TYPE ST_OutputStationHSSustainabilityData :
STRUCT
	{attribute 'OPC.UA.DA.Description' := 'Dummy (for making struct visible on OPC UA'}
	bDummy						: BOOL;
END_STRUCT
END_TYPE

(* stored: Version 1.1.0.1, ProductVersion 3.1.4024.2
   DUT ST_OutputStationHSSustainabilityData: Id {675205f0-53fc-4d1a-8f9a-a940df424982} *)
